PROGRAM MAIN

VAR
	
END_VAR

//Milan Oude Nijeweme
//517922
//Process and Safety individual assignment

//This program provides a structured morning routine where, in sequence, an alarm goes off,
//lights turn on, and coffee is made. it accounts for the day of the week to determine if
//it's a workday and includes a reset feature to restore all actions and prepare for the
//next routine.


//Ceck if the alarm is set and is currently off
IF GVL.bSetAlarm AND NOT GVL.bAlarmON THEN
		GVL.AlarmTimer(IN := TRUE, PT := GVL.AlarmTime); //Starts the timer for the alarm with the predefined time
			IF GVL.AlarmTimer.Q THEN
				GVL.bAlarmON := TRUE;
		 
				GVL.DayCounter := GVL.DayCounter + 1; //Keeps track of day changes
		
					IF GVL.DayCounter > 7 THEN //Reset DayCounter to 1 if it exceeds 7 so its a weekly cycle
						GVL.DayCounter := 1;
					END_IF
			
				GVL.AlarmTimer(IN := FALSE);
				gvl.bSetAlarm := FALSE;	
			END_IF
END_IF

//Determine if it's a workday based on the current day
GVL.bWorkDayStatus := IsItAWorkDay(GVL.DayCounter);



//Gives the name of the day 
GVL.TheDayOfWeek := DayOfWeek(GVL.DayCounter);

//Light activation
LightsON();

//Resets all the variables so the alarm can be set again.
IF GVL.bReset THEN
	GVL.ResetTimer(IN:=TRUE, PT := T#1S);
	IF GVL.ResetTimer.Q THEN
		GVL.bAlarmON := FALSE;
		GVL.bLightsON := FALSE;
		GVL.bCoffeeReady := FALSE;
		GVL.bReset := FALSE;
		GVL.ResetTimer(IN:=FALSE);
	END_IF
	
END_IF

END_PROGRAM

(* stored: Version 1.1.0.1, ProductVersion 3.1.4024.12
   POU MAIN: Id {cd2eb92e-b13a-41b7-9c9e-feae7366627f}, SpecialFunc None *)
